# B&R Automation Studio project lab1_git
Automation Studio 4.5.2.102

## Configuration Config1

### Task classes (Cpu.sw)
```
Cyclic#1:
  Program <- Program.prg
Libraries: TEMALAB1
```

## Logical view

Binary libraries used (declarations not repeated): operator, runtime, astime, AsIecCon

### Library Logical/Libraries/TEMALAB1 (ANSIC)

#### FB_motor.c
```c
#include <bur/plctypes.h>
#ifdef __cplusplus
	extern "C"
	{
#endif
	#include "TEMALAB1.h"
#ifdef __cplusplus
	};
#endif
/* TODO: Add your comment here */
void FB_Motor(struct FB_Motor* inst)
{
	REAL a = (inst->u/inst->ke) - inst->w;
	REAL b = a / inst->Tm;

	inst->integrator.in = b;
	FB_Integrator(&inst->integrator);

	inst->w = inst->integrator.out;

	inst->integrator.in = inst->w;
	FB_Integrator(&inst->integrator);

	inst->phi = inst->integrator.out;

}
```

#### FB_Integrator.c
```c
#include <bur/plctypes.h>
#ifdef __cplusplus
	extern "C"
	{
#endif
	#include "TEMALAB1.h"
#ifdef __cplusplus
	};
#endif
/* TODO: Add your comment here */
void FB_Integrator(struct FB_Integrator* inst)
{
	inst->dt = d_t;
	inst->out = inst->dt * inst->in + inst->prev_value;
	inst->prev_value = inst->out;
}
```

#### FB_Controller.c
```c
#include <bur/plctypes.h>
#ifdef __cplusplus
	extern "C"
	{
#endif
	#include "TEMALAB1.h"
#ifdef __cplusplus
	};
#endif
/* TODO: Add your comment here */
void FB_Controller(struct FB_Controller* inst)
{
	REAL a = inst->e_in * inst->k_p;
	REAL b = inst->e_in * inst->k_i;

	a = a > inst->max_abs_value ? inst->max_abs_value : a;
	a = a < -inst->max_abs_value ? -inst->max_abs_value : a;

	inst->integrator.in = b + inst->last_sum;
	FB_Integrator(&inst->integrator);

	REAL sum = a + inst->integrator.out;

	inst->u_out = sum;//inst->u_out = inst->a

	inst->u_out = inst->u_out > inst->max_abs_value ? inst->max_abs_value : inst->u_out;
	inst->u_out = inst->u_out < -inst->max_abs_value ? -inst->max_abs_value : inst->u_out;

	inst->last_sum = inst->u_out - sum; //inst->iyOld = inst->u_out - sum;

}
```

### Program Logical/Program

#### Variables.var
```iecst
VAR
	enable : BOOL;
	counter : {REDUND_UNREPLICABLE} UINT;
	speed : {REDUND_UNREPLICABLE} REAL;
	fb_motor2 : FB_Motor;
	fb_motor1 : FB_Motor;
	fb_controller : FB_Controller;
	integrator : FB_Integrator;
END_VAR
```

#### Main.c
```c
#include <bur/plctypes.h>

#ifdef _DEFAULT_INCLUDES
	#include <AsDefault.h>
#endif

void _INIT ProgramInit(void)
{
	fb_motor1.ke = 0.0735;
	fb_motor1.Tm = 0.147;
	fb_motor1.u = 0;
	fb_motor1.dt = 0.01;

	fb_motor2.ke = 0.0735;
	fb_motor2.Tm = 0.147;
	fb_motor2.u = 0;
	fb_motor2.dt = 0.01;

	fb_controller.k_p = 0.108045;
	fb_controller.k_i = 0.735;
	fb_controller.max_abs_value = 24.0;
	fb_controller.dt = 0.01;

	speed = 0;
	counter = 0;
	enable = 1;
}

void _CYCLIC ProgramCyclic(void)
{
	if(enable)
	{
		if(counter == 200)
		{
			speed = 0;
			counter = 0;
		}
		else if (counter == 50)
		{
			speed = 50;
		}

		fb_controller.e_in = speed - fb_motor1.w;
		FB_Controller(&fb_controller);

		fb_motor1.u = fb_controller.u_out;
		FB_Motor(&fb_motor1);

		fb_motor2.u = speed * fb_motor2.ke;
		FB_Motor(&fb_motor2);

		counter++;
	}
}

void _EXIT ProgramExit(void)
{

}
```

Listed in the project but not available here: Logical/Libraries/TEMALAB1/Types.typ, Logical/Libraries/TEMALAB1/Constants.var, Logical/Libraries/TEMALAB1/TEMALAB1.fun
